{attribute 'qualified_only'}
VAR_GLOBAL CONSTANT
	// Mirrors Beckhoff's own Global_Version.stLibVersion_* pattern (see ST_LibVersion),
	// which only covers Tc2_*/Tc3_* library references, not custom ones -- until now: this
	// GVL uses Beckhoff's own naming exactly, so it merges into a consumer's Global_Version.
	// Kept in sync with <ProjectVersion> in MONETNRuntime.plcproj at release time.
	// SA0033 (unused variable) is a hard error in this project; this constant is meant
	// to be read externally via ADS, never referenced internally, so it's suppressed here.
	{attribute 'analysis' := '-33'}
	stLibVersion_MONETNRuntime : ST_LibVersion := (
		iMajor := 0,
		iMinor := 1,
		iBuild := 2,
		iRevision := 0,
		nFlags := 1,
		sVersion := '0.1.2'
	);
END_VAR

(* stored: Version 1.1.0.1, ProductVersion 3.1.4024.15
   GVL Global_Version: Id {862891c1-e7c0-4d93-9d29-123b9e39cac0} *)
